(* IEC 61131-3 sources: RL_MAR/experiments/comparison/autoplc/results/gpt-4o_20260511_211137/med_69, 1 file *)

(* ---- med_69_1.st ---- *)
FUNCTION_BLOCK FB_ValueOut
    VAR_INPUT
        valueIn : INT;
        conf : UINT;
    END_VAR

    VAR_OUTPUT
        ValueOut : INT;
    END_VAR

    VAR
        tempValue : INT;
    END_VAR

    // Initialization
    ValueOut := 0;

    // Configuration Handling
    CASE conf OF
        1, 2:
            // Divide valueIn by 10
            tempValue := valueIn / 10;
            IF tempValue < 0 THEN
                ValueOut := 0;
            ELSE
                ValueOut := tempValue;
            END_IF;
        3:
            // Specific mappings for valueIn
            CASE valueIn OF
                0:
                    ValueOut := 0;
                300:
                    ValueOut := 163;
                600:
                    ValueOut := 331;
                ELSE
                    ValueOut := 0;
            END_CASE;
        6, 7:
            // Specific mappings for valueIn
            IF valueIn = 100 THEN
                ValueOut := 319;
            ELSE
                ValueOut := 0;
            END_IF;
        4, 5, 8, 9, 10:
            // Default behavior for unspecified configurations
            ValueOut := 0;
        ELSE
            // Default behavior for unspecified configurations
            ValueOut := 0;
    END_CASE;
END_FUNCTION_BLOCK
